Universal Robots PolyScope program: IAC000 Vision Test.urp

Program IAC000 Vision Test (installation=default directory=/programs createdIn=5.9.1.1031110 lastSavedIn=5.9.1.1031110 robotSerialNumber=20195501059)
Calibrated DH parameters: a=[0.000146, -0.418764, -0.053981, 0.000058, -0.000023, 0]; d=[0.162545, 37.319448, -206.067439, 168.881546, 0.09955, 0.099464]; alpha=[1.57004, -0.001979, 0.002304, 1.570607, -1.57066, 0]; deltaTheta=[0, -0.174616, -1.258233, 1.432844, -0.000001, 0]
BeforeStart
  URCap Gripper Activate (Robotiq_Grippers, Robotiq Inc.) dataModel(ResetAndActivateKey=false)
  initial_p := get_actual_tcp_pose()
  MoveJ speed 60 deg/s, acceleration 80 deg/s^2 (useActiveTCP=true) feature=Base
    Waypoint Waypoint (Variable): variable=initial_p
Robot Program (runOnlyOnce=false)
  URCap Gripper (Robotiq_Grippers, Robotiq Inc.) dataModel(position=100.0, force=100.0, speed=100.0, positionInDouble=100.0, forceInDouble=100.0, speedInDouble=100.0, slaveIds=[9], blocking=true)
  MoveL speed 250 mm/s, acceleration 1200 mm/s^2 (useActiveTCP=true) feature=Base
    Waypoint home: TCP in base x=353.442 y=-425.051 z=15.364 mm, rx=-2.1827 ry=-2.2594 rz=0 rad; joints [115.734, -68.978, 112.532, -133.544, 270.037, 113.795] deg; TCP offset x=0 y=0 z=174 mm, rx=0 ry=0 rz=0 rad
  Call vision_connect
  Loop Forever
    MoveL speed 250 mm/s, acceleration 1200 mm/s^2 (useActiveTCP=true) feature=Base
      Waypoint calibrate_pose: TCP in base x=251.976 y=-487.932 z=207.251 mm, rx=1.1672 ry=2.7547 rz=-0.3884 rad; joints [104.95, -89.901, 111.676, -127.845, 266.662, 60.419] deg
    Call vision_acquire_only
  Call vision_disconnect
SubProgram  [hidden by the author, left out]
SubProgram  [hidden by the author, left out]
SubProgram  [hidden by the author, left out]
SubProgram vision_read_barcode [hidden by the author, left out]
SubProgram vision_connect [hidden by the author, left out]
SubProgram vision_acquire_only [hidden by the author, left out]
SubProgram vision_disconnect [hidden by the author, left out]
